// LS Electric XG5000 project: PLC 시험2
// PLC LSPLC
// module base 0 slot 0: 입출력 모듈:XBC-DR14E (DC 24V 입력 8점, 릴레이 출력 6점)

PROGRAM NewProgram (task: 스캔 프로그램)

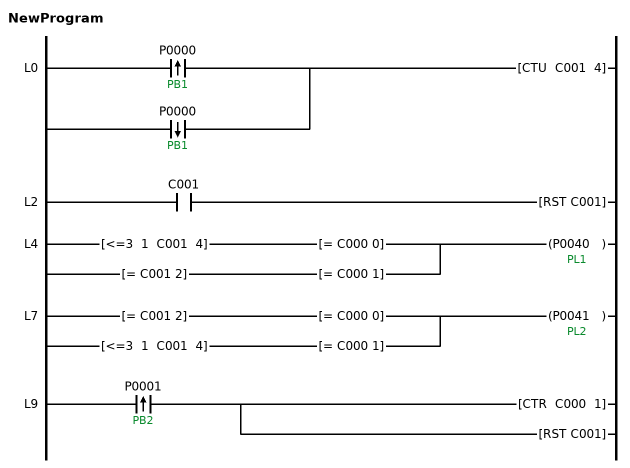
; L0
LOADP     P0000	// PB1
ORN       P0000	// PB1
CTU       C001 4
; L2
LOAD      C001
RST       C001
; L4
LOAD<=3   1 C001 4
AND=      C000 0
LOAD=     C001 2
AND=      C000 1
OR LOAD
OUT       P0040	// PL1
; L7
LOAD=     C001 2
AND=      C000 0
LOAD<=3   1 C001 4
AND=      C000 1
OR LOAD
OUT       P0041	// PL2
; L9
LOADP     P0001	// PB2
CTR       C000 1
RST       C001

VARIABLES AND COMMENTS (devices not used above)
P00002	BIT	PB3